(* PLC project Programme MGS_2-07_refactorJOY.project, CODESYS CODESYS V3.5 SP19 Patch 1 *)
(* stored: creationDateTime 2026-06-29T23:37:40.1406681, modificationDateTime 2026-06-29T22:49:33.424 *)

PROGRAM diagCAN
  VAR
    BusState : BUS_STATE;  (* Bus & Device states *)
    DeviceState : DEVICE_STATE;
    BusError : INT;  (* Internal function execution errors (0 = NO_ERROR) *)
    DeviceError : INT;
    BusDiagAvailable : BOOL;  (* Diagnosis status flags *)
    DevDiagAvailable : BOOL;
    IsOnline : BOOL;  (* Device is physically present on the bus *)
    IsOperational : BOOL;  (* Device is running and actively processing I/O (PDO) *)
  END_VAR

            // 1. Get CAN bus logic status
BusState := CANopen_Manager.GetBusState(
    xDiagnosisInfoAvailable => BusDiagAvailable, 
    eError => BusError
);

// 2. Get Joystick node status
DeviceState := JOY1_JOYSTICK_MCB560_CO4201A.GetDeviceState(
    xDiagnosisInfoAvailable => DevDiagAvailable, 
    eError => DeviceError
);

// 3. Evaluate if device is physically connected/found
IF DeviceState <> DEVICE_STATE.NOT_FOUND THEN
    IsOnline := TRUE;
ELSE
    IsOnline := FALSE;
END_IF;

// 4. Evaluate if device is actively Operational (NMT Operational / Running)
IF DeviceState = DEVICE_STATE.RUNNING THEN
    IsOperational := TRUE;
ELSE
    IsOperational := FALSE; 
    // (If FALSE, it might be stopped, pre-operational, or disconnected)
END_IF;
          
END_PROGRAM
